// TIA Portal V18 export
// export: Created 2026-01-09T11:31:57.0910137Z, ExportSetting WithDefaults, DisplayName Totally Integrated Automation Portal, DisplayVersion V18 Update 5, DisplayName TIA Portal Openness, DisplayVersion V18 Update 5, DisplayName TIA Portal Teamcenter Gateway, DisplayVersion V18, DisplayName TIA Portal Version Control Interface, DisplayVersion V18, DisplayName SINAMICS Startdrive Advanced, DisplayVersion V18 SP2 Update 1, DisplayName SINAMICS Startdrive G110M, G120, G120C, G120D, G120P, G115D, DisplayVersion V18 SP2 Update 1, DisplayName SINAMICS Startdrive G130, G150, S120, S150, SINAMICS MV, S210, G220, S200, DisplayVersion V18 SP2 Update 1, DisplayName STEP 7 Professional, DisplayVersion V18 Update 5, DisplayName STEP 7 Safety, DisplayVersion V18, DisplayName WinCC Professional, DisplayVersion V18 Update 5
TagTable "ST350_Recpie"
  RecipeDB_ParameterElement_TypeID : USInt  (PLC tag ST10_RecipeDB.ParameterElement.TypeID, CPU S71500-2PN_TP700, 1 s)
  RecipeDB_ParameterElement_TypeName : String  (PLC tag ST10_RecipeDB.ParameterElement.TypeName, CPU S71500-2PN_TP700, 1 s)
  STxxx_RecipeDB_ParameterElement_FixtureID{1} : Byte  (PLC tag ST10_RecipeDB.ParameterElement.FixtureID[1], CPU S71500-2PN_TP700, 1 s)
  Spare : WString  (1 s)
  ST10_RecipeDB_ParameterElement_A1_TableFixtureCode : Array [0..10] of String  (PLC tag ST10_RecipeDB.ParameterElement.A1_TableFixtureCode, CPU S71500-2PN_TP700, 1 s)
    TagArrayMember "[0]"
    TagArrayMember "[1]"
    TagArrayMember "[2]"
    TagArrayMember "[3]"
    TagArrayMember "[4]"
    TagArrayMember "[5]"
    TagArrayMember "[6]"
    TagArrayMember "[7]"
    TagArrayMember "[8]"
    TagArrayMember "[9]"
    TagArrayMember "[10]"
  ST10_RecipeDB_ParameterElement_A2_TableFixtureCode : Array [0..10] of String  (PLC tag ST10_RecipeDB.ParameterElement.A2_TableFixtureCode, CPU S71500-2PN_TP700, 1 s)
    TagArrayMember "[0]"
    TagArrayMember "[1]"
    TagArrayMember "[2]"
    TagArrayMember "[3]"
    TagArrayMember "[4]"
    TagArrayMember "[5]"
    TagArrayMember "[6]"
    TagArrayMember "[7]"
    TagArrayMember "[8]"
    TagArrayMember "[9]"
    TagArrayMember "[10]"
  ST10_RecipeDB_ParameterElement_A1RingUnloadingFixtureCode : String  (PLC tag ST10_RecipeDB.ParameterElement.A1RingUnloadingFixtureCode, CPU S71500-2PN_TP700, 1 s)
  ST10_RecipeDB_ParameterElement_E1LoadingNGFixtureCode : String  (PLC tag ST10_RecipeDB.ParameterElement.E1LoadingNGFixtureCode, CPU S71500-2PN_TP700, 1 s)
  ST10_RecipeDB_ParameterElement_ShaftScanFixtureCode : String  (PLC tag ST10_RecipeDB.ParameterElement.ShaftScanFixtureCode, CPU S71500-2PN_TP700, 1 s)
  ST10_RecipeDB_ParameterElement_B1PressFixtureCode : String  (PLC tag ST10_RecipeDB.ParameterElement.B1PressFixtureCode, CPU S71500-2PN_TP700, 1 s)
  ST10_RecipeDB_ParameterElement_CGlueFixtureCode : String  (PLC tag ST10_RecipeDB.ParameterElement.CGlueFixtureCode, CPU S71500-2PN_TP700, 1 s)
  ST10_RecipeDB_ParameterElement_B1PressCylFixtureCode : String  (PLC tag ST10_RecipeDB.ParameterElement.B1PressCylFixtureCode, CPU S71500-2PN_TP700, 1 s)
  ST10_RecipeDB_ParameterElement_A2RingUnloadingFixtureCode : String  (PLC tag ST10_RecipeDB.ParameterElement.A2RingUnloadingFixtureCode, CPU S71500-2PN_TP700, 1 s)
  ST10_RecipeDB_ParameterElement_E2UnloadingNGFixtureCode : String  (PLC tag ST10_RecipeDB.ParameterElement.E2UnloadingNGFixtureCode, CPU S71500-2PN_TP700, 1 s)
  ST10_RecipeDB_ParameterElement_B2PressFixtureCode : String  (PLC tag ST10_RecipeDB.ParameterElement.B2PressFixtureCode, CPU S71500-2PN_TP700, 1 s)
  ST10_RecipeDB_ParameterElement_CGlueNGFixtureCode : String  (PLC tag ST10_RecipeDB.ParameterElement.CGlueNGFixtureCode, CPU S71500-2PN_TP700, 1 s)
  ST10_RecipeDB_ParameterElement_B2PressCylFixtureCode : String  (PLC tag ST10_RecipeDB.ParameterElement.B2PressCylFixtureCode, CPU S71500-2PN_TP700, 1 s)
  ST10_RecipeDB_ParameterElement_B1PressProgram : Int  (PLC tag ST10_RecipeDB.ParameterElement.B1PressProgram, CPU S71500-2PN_TP700, 1 s)
  ST10_RecipeDB_ParameterElement_B2PressProgram : Int  (PLC tag ST10_RecipeDB.ParameterElement.B2PressProgram, CPU S71500-2PN_TP700, 1 s)
  ST10_RecipeDB_ParameterElement_CGlueShaftIV3Program_1 : Word  (PLC tag ST10_RecipeDB.ParameterElement.CGlueShaftIV3Program_1, CPU S71500-2PN_TP700, 1 s)
  ST10_RecipeDB_ParameterElement_CGlueShaftIV3Program_2 : Word  (PLC tag ST10_RecipeDB.ParameterElement.CGlueShaftIV3Program_2, CPU S71500-2PN_TP700, 1 s)
  ST10_RecipeDB_ParameterElement_CGlueShaftIV3Program_3 : Word  (PLC tag ST10_RecipeDB.ParameterElement.CGlueShaftIV3Program_3, CPU S71500-2PN_TP700, 1 s)
  ST10_RecipeDB_ParameterElement_CGlueShaftIV3Program_4 : Word  (PLC tag ST10_RecipeDB.ParameterElement.CGlueShaftIV3Program_4, CPU S71500-2PN_TP700, 1 s)
  ST10_RecipeDB_ParameterElement_CGlueMagnetIV3Program : Word  (PLC tag ST10_RecipeDB.ParameterElement.CGlueMagnetIV3Program, CPU S71500-2PN_TP700, 1 s)
  ST10_RecipeDB_ParameterElement_CGlueProgram : Int  (PLC tag ST10_RecipeDB.ParameterElement.CGlueProgram, CPU S71500-2PN_TP700, 1 s)
  AutoProcessData_Gripper1_LCode_R1[1] : String  (PLC tag AutoProcessData.GripperCode_R1[1], CPU S71500-2PN_TP700, 1 s)
  AutoProcessData_Gripper1_RCode_R1[2] : String  (PLC tag AutoProcessData.GripperCode_R1[2], CPU S71500-2PN_TP700, 1 s)
  AutoProcessData_Gripper2_LCode_R1[3] : String  (PLC tag AutoProcessData.GripperCode_R1[3], CPU S71500-2PN_TP700, 1 s)
  AutoProcessData_Gripper2_RCode_R1[4] : String  (PLC tag AutoProcessData.GripperCode_R1[4], CPU S71500-2PN_TP700, 1 s)
  AutoProcessData_Gripper1_LCode_R2[1] : String  (PLC tag AutoProcessData.GripperCode_R2[1], CPU S71500-2PN_TP700, 1 s)
  AutoProcessData_Gripper1_RCode_R2[2] : String  (PLC tag AutoProcessData.GripperCode_R2[2], CPU S71500-2PN_TP700, 1 s)
  AutoProcessData_Gripper2_LCode_R2[3] : String  (PLC tag AutoProcessData.GripperCode_R2[3], CPU S71500-2PN_TP700, 1 s)
  AutoProcessData_Gripper2_RCode_R2[4] : String  (PLC tag AutoProcessData.GripperCode_R2[4], CPU S71500-2PN_TP700, 1 s)
  AutoProcessData_Gripper1_LCode_R3[1] : String  (PLC tag AutoProcessData.GripperCode_R3[1], CPU S71500-2PN_TP700, 1 s)
  AutoProcessData_Gripper1_RCode_R3[2] : String  (PLC tag AutoProcessData.GripperCode_R3[2], CPU S71500-2PN_TP700, 1 s)
  AutoProcessData_Gripper2_LCode_R3[3] : String  (PLC tag AutoProcessData.GripperCode_R3[3], CPU S71500-2PN_TP700, 1 s)
  AutoProcessData_Gripper2_RCode_R3[4] : String  (PLC tag AutoProcessData.GripperCode_R3[4], CPU S71500-2PN_TP700, 1 s)
  ST10_RecipeDB_ParameterElement_R1GripperFixtureCode : Array [0..6] of String  (PLC tag ST10_RecipeDB.ParameterElement.R1GripperFixtureCode, CPU S71500-2PN_TP700, 1 s)
    TagArrayMember "[0]"
    TagArrayMember "[1]"
    TagArrayMember "[2]"
    TagArrayMember "[3]"
    TagArrayMember "[4]"
    TagArrayMember "[5]"
    TagArrayMember "[6]"
  ST10_RecipeDB_ParameterElement_R2GripperFixtureCode : Array [0..6] of String  (PLC tag ST10_RecipeDB.ParameterElement.R2GripperFixtureCode, CPU S71500-2PN_TP700, 1 s)
    TagArrayMember "[0]"
    TagArrayMember "[1]"
    TagArrayMember "[2]"
    TagArrayMember "[3]"
    TagArrayMember "[4]"
    TagArrayMember "[5]"
    TagArrayMember "[6]"
  ST10_RecipeDB_ParameterElement_R3GripperFixtureCode : Array [0..6] of String  (PLC tag ST10_RecipeDB.ParameterElement.R3GripperFixtureCode, CPU S71500-2PN_TP700, 1 s)
    TagArrayMember "[0]"
    TagArrayMember "[1]"
    TagArrayMember "[2]"
    TagArrayMember "[3]"
    TagArrayMember "[4]"
    TagArrayMember "[5]"
    TagArrayMember "[6]"
